# B&R Automation Studio project MM_movim_manuale (part 2)

```c
		if (inst->gs.st_ninfo == 0)																						/* if returned value ok...		*/
		{
			VAL_TO_ASCII(inst->gs.data_typ, inst->gs.ascii_value, inst->gs.var_addr);									/* convert from num to ascii value	*/

			strcpy ( (USINT *)inst->mem_part_all.mem + inst->offset, &inst->gs.name[0]);
			inst->offset = strlen((USINT *) inst->mem_part_all.mem);													/* calculate actual buffer legth	*/
			BUFFER(inst->offset) = inst->chr_separ;																		/* put char separator 			*/
			inst->offset = inst->offset + 1;																			/* calculate actual buffer legth	*/

			inst->get_comm.enable = 1;																					/* enable fub				*/
			Rec_get_comm(&inst->get_comm);																				/* call fub					*/

			if ((inst->get_comm.status == 0) || (inst->get_comm.status == 1))											/* if status ok...			*/
			{
				strcpy ( (USINT *)inst->mem_part_all.mem + inst->offset, &inst->get_comm.comm[0]);						/* ...copy comment			*/
				inst->offset = strlen((USINT *) inst->mem_part_all.mem);												/* calculate actual buffer legth	*/
				BUFFER(inst->offset) = inst->chr_separ;																	/* put char separator 			*/
				inst->offset = inst->offset + 1;																		/* calculate actual buffer legth	*/
			}
			else																										/* if error occurred...			*/
			{
				SET_ERROR(inst->get_comm.status);																		/* ... go to error step			*/
			}
			strcpy ( (USINT *)inst->mem_part_all.mem + inst->offset, inst->gs.ascii_value);								/* copy value (in ascii format)	*/
			inst->offset = strlen((USINT *) inst->mem_part_all.mem);													/* calculate actual buffer legth	*/
			BUFFER(inst->offset    ) = 13;																				/* put carriage return 			*/
			BUFFER(inst->offset + 1) = 10; 																				/* put line feed 				*/
 			inst->offset = inst->offset = inst->offset + 2;																/* calculate actual buffer legth	*/

			memset(&inst->gs.ascii_value, 0, sizeof (inst->gs.ascii_value));											/* reset ascii value buffer		*/

			if (inst->gs.dim[inst->gs.idx_lev] > 1)																		/* if dim > 0 it's an array... 	*/
			{
				clear(&inst->gs.name[0], '[');																			/* ...then delete square brackets 	*/
			}
			if (inst->gs.cnt_dim[inst->gs.idx_lev] < inst->gs.dim[inst->gs.idx_lev] )      								/* if not last element of array... 	*/
			{
				inst->gs.cnt_dim[inst->gs.idx_lev]++;																	/* ...increment index-counter		*/
			}

			for (inst->k = inst->gs.idx_lev;  (inst->gs.cnt_dim[inst->k] == inst->gs.dim[inst->k] && (inst->gs.idx_lev > 0) ); inst->k--)
			{
			 	if (inst->gs.flag_arr_str[inst->k - 1] == 1)															/* if it's an array of structures...*/
				{
					clear(&inst->gs.name[0], '[');																		/* ...delete square brackets		*/
					inst->gs.cnt_arr_str[inst->k-1]++;																	/* increment array of struct counter*/
					if (inst->gs.cnt_arr_str[inst->k-1] >= inst->gs.dim[inst->k - 1] )									/* if array of struct's last element*/
					{
						inst->gs.cnt_arr_str[inst->k-1] = 0;															/* ... reset counter			*/
					}
				}
				else																									/* if field isn't array of structs..*/
				{
					clear(&inst->gs.name[0], '.');																		/* ..delete field name			*/
				}
				inst->gs.cnt_dim[inst->k] = 0;																			/* reset counter for this level	*/
				inst->gs.cnt_dim[inst->k-1] ++;																			/* go ahead for previous level	*/
				inst->gs.idx_lev--;																						/* decrement level 			*/
			}

			if ((inst->gs.idx_lev == 0) &&(inst->gs.cnt_dim[0] == inst->gs.dim[0]))										/* this is the end-condition 		*/
			{
				for (inst->k = 0; inst->k < DEEP_STR; inst->k++)														/* scan all struct (tree)		*/
				{
					inst->gs.cnt_dim[inst->k] = 0;																		/* reset counters about dimensions	*/
					inst->gs.dim[inst->k]     = 0;																		/* reset dimensions			*/
				}
				inst->step = STEP_WST_WRITE_DATA;																		/* ...go again to previous step	*/
			}
			else																										/* if write procedure not finished..*/
			{
				inst->step = STEP_WST_INFO_DATA;																		/* ...go again to previous step	*/
			}
		}
		else																											/* if error occurred...			*/
		{
			SET_ERROR(inst->gs.st_ninfo);																				/* ...go to error step			*/
		}
	}
	else																												/* if error occurred...			*/
	{
	 	SET_ERROR(inst->gs.ret_pvixgetadr);																				/* ...go to error step			*/
	}

} /* end Write_data() */
```

#### Recipe.fun
```iecst
FUNCTION_BLOCK Rec_get_comm
VAR
		step	:USINT;
		k	:UDINT;
		j	:UDINT;
		start	:UDINT;
		do_info	:DatObjInfo;
		count_comm	:UDINT;
		prevstep	:USINT;
	END_VAR
	VAR_INPUT
		enable	:BOOL;
	END_VAR
	VAR_OUTPUT
		comm	:STRING[45];
		status	:UINT;
	END_VAR
END_FUNCTION_BLOCK
FUNCTION_BLOCK Rec_Write
VAR
		overw	:USINT;
		recipecsv	:STRING[24];
		chr_separ	:USINT;
		firstrow_written	:BOOL;
		step	:USINT;
		k	:UDINT;
		fileio_id	:UDINT;
		offset	:UDINT;
		gs	:gs_typ;
		get_comm	:Rec_get_comm;
		FOpen	:FileOpen;
		FCreate	:FileCreate;
		FClose	:FileClose;
		FWrite	:FileWrite;
		FDelete	:FileDelete;
		get_sys_err	:UINT;
		prevstep	:USINT;
		repeat_switch	:USINT;
		mem_part_all	:AsMemPartAlloc;
		mem_allocated	:BOOL;
		mem_part_free	:AsMemPartFree;
		limit_repeat_cntr	:USINT;
		tmp_status	:UINT;
	END_VAR
	VAR_INPUT
		enable	:BOOL;
		structure	:STRING[15];
		recipe	:STRING[20];
		ident	:UDINT;
		speed_option	:BOOL;
	END_VAR
	VAR_OUTPUT
		status	:UINT;
		msg_err	:STRING[80];
	END_VAR
END_FUNCTION_BLOCK
FUNCTION_BLOCK Rec_NameRead
VAR
		step	:USINT;
		set_device	:USINT;
		DInfo	:DirInfo;
		DRead	:DirRead;
		ReadData	:fiDIR_READ_DATA;
		get_sys_err	:UINT;
		prevstep	:USINT;
		len_name	:UINT;
		file_counter	:UDINT;
		tot_files	:UDINT;
		not_valid_csv	:USINT;
	END_VAR
	VAR_INPUT
		enable	:BOOL;
	END_VAR
	VAR_OUTPUT
		status	:UINT;
		msg_err	:STRING[80];
		recipe	:STRING[20];
		nr_csv_read	:UDINT;
	END_VAR
END_FUNCTION_BLOCK
FUNCTION_BLOCK Rec_Import
VAR
		step	:USINT;
		get_sys_err	:UINT;
		prevstep	:UINT;
		recipecsv	:STRING[24];
		FCopy	:FileCopy;
	END_VAR
	VAR_INPUT
		enable	:BOOL;
		recipe	:STRING[20];
	END_VAR
	VAR_OUTPUT
		status	:UINT;
		msg_err	:STRING[80];
	END_VAR
END_FUNCTION_BLOCK
FUNCTION_BLOCK Rec_Imp_All
VAR
		recipe	:STRING[260];
		read_name	:Rec_NameRead;
		rec_imp	:Rec_Import;
		step	:USINT;
		get_sys_err	:UINT;
		prevstep	:USINT;
	END_VAR
	VAR_INPUT
		enable	:BOOL;
	END_VAR
	VAR_OUTPUT
		status	:UINT;
		msg_err	:STRING[80];
		nr_csv_imported	:UDINT;
		recipe_imp	:STRING[80];
	END_VAR
END_FUNCTION_BLOCK
FUNCTION_BLOCK Rec_Export
VAR
		step	:USINT;
		get_sys_err	:UINT;
		prevstep	:UINT;
		recipecsv	:STRING[24];
		FCopy	:FileCopy;
	END_VAR
	VAR_INPUT
		enable	:BOOL;
		recipe	:STRING[20];
	END_VAR
	VAR_OUTPUT
		status	:UINT;
		msg_err	:STRING[80];
	END_VAR
END_FUNCTION_BLOCK
FUNCTION_BLOCK Rec_Exp_All
VAR
		recipe	:STRING[260];
		read_name	:Rec_NameRead;
		rec_exp	:Rec_Export;
		step	:USINT;
		get_sys_err	:UINT;
		prevstep	:USINT;
	END_VAR
	VAR_INPUT
		enable	:BOOL;
	END_VAR
	VAR_OUTPUT
		status	:UINT;
		msg_err	:STRING[80];
	END_VAR
END_FUNCTION_BLOCK
FUNCTION_BLOCK Rec_Upload
VAR
		recipecsv	:STRING[24];
		step	:USINT;
		offset	:UDINT;
		k	:UDINT;
		j	:UDINT;
		ascii_infile	:ARRAY [0..21] OF USINT;
		gs	:gs_typ;
		FOpen	:FileOpen;
		FRead	:FileRead;
		FClose	:FileClose;
		get_sys_err	:UINT;
		repeat_switch	:USINT;
		prevstep	:USINT;
		mem_part_all	:AsMemPartAlloc;
		mem_allocated	:BOOL;
		mem_part_free	:AsMemPartFree;
		limit	:USINT;
		tmp_status	:UINT;
	END_VAR
	VAR_INPUT
		enable	:BOOL;
		structure	:STRING[15];
		recipe	:STRING[20];
		ident	:UDINT;
		speed_option	:BOOL;
	END_VAR
	VAR_OUTPUT
		status	:UINT;
		msg_err	:STRING[80];
	END_VAR
END_FUNCTION_BLOCK
FUNCTION_BLOCK Rec_Delete
VAR
		recipecsv	:STRING[24];
		step	:USINT;
		FDelete	:FileDelete;
		get_sys_err	:UINT;
		prevstep	:USINT;
	END_VAR
	VAR_INPUT
		enable	:BOOL;
		recipe	:STRING[20];
	END_VAR
	VAR_OUTPUT
		status	:UINT;
		msg_err	:STRING[80];
	END_VAR
END_FUNCTION_BLOCK
FUNCTION_BLOCK Rec_Init
VAR
		step	:USINT;
		dir_create	:DirCreate;
		prevstep	:USINT;
		mem_part_create	:AsMemPartCreate;
	END_VAR
	VAR_INPUT
		enable	:BOOL;
	END_VAR
	VAR_OUTPUT
		ident	:UDINT;
		status	:UINT;
		msg_err	:STRING[80];
	END_VAR
END_FUNCTION_BLOCK
```

- Visualisation Logical/Visu (not shown)

### Program Logical/Program (ANSIC)

#### Variables.var
```iecst
VAR
	Apertura_T : BOOL;
	Alta_V_TON : TON;
	Ap_TON : TON;
	Ch_TON : TON;
	Alta_velocita_T : BOOL;
	Chiusura_T : BOOL;
END_VAR
```

#### Cyclic.c
```c
#include <bur/plctypes.h>

#ifdef _DEFAULT_INCLUDES
	#include <AsDefault.h>
#endif

#define CONVERT_INT_TO_ANA_1(x, x1, y1, x2, y2)  ( y1 + ( (y2 - y1) / (REAL) (x2 - x1) ) * (x - x1) )

void _CYCLIC ProgramCyclic(void)
{
	glb_io.Ai.oil_pressure_conv           		= (CONVERT_INT_TO_ANA_1(glb_io.Ai.oil_pressure,           		0,  0, 32767, 250));
	glb_io.Ai.p_apertura_conv           		= (CONVERT_INT_TO_ANA_1(glb_io.Ai.p_apertura,           		0,  0, 32767, 250));
	glb_io.Ai.p_chiusura_conv           		= (CONVERT_INT_TO_ANA_1(glb_io.Ai.p_chiusura,           		0,  0, 32767, 250));

	Report.oil_pressure		= glb_io.Ai.oil_pressure_conv;
	Report.p_apertura		= glb_io.Ai.p_apertura_conv;
	Report.p_apertura		= glb_io.Ai.p_chiusura_conv;

	// ritardo attivazione alta velocità //
	if (hmi.cmd.alta_velocita){
		Alta_V_TON.IN = (hmi.cmd.apertura || hmi.cmd.chiusura);
		Alta_V_TON.PT = 1500;
		TON(&Alta_V_TON);
		Alta_velocita_T = Alta_V_TON.Q;
	} else {
		Alta_velocita_T = 0;
	}
	glb_io.out.alta_velocita = Alta_velocita_T;

	// ritardo attivazione apertura //
	Ap_TON.IN = hmi.cmd.apertura;
	Ap_TON.PT = 500;
	TON(&Ap_TON);
	Apertura_T = Ap_TON.Q;

	// ritardo attivazione chiusura //
	Ch_TON.IN = hmi.cmd.chiusura;
	Ch_TON.PT = 500;
	TON(&Ch_TON);
	Chiusura_T = Ch_TON.Q;

	// COMANDI //
	// SCARICO PRESSIONE //
	if (hmi.cmd.chiusura || hmi.cmd.scarico_ap) glb_io.out.Scarico_ap = 1; else glb_io.out.Scarico_ap = 0;
	if (hmi.cmd.apertura || hmi.cmd.scarico_ch) glb_io.out.Scarico_ch = 1; else glb_io.out.Scarico_ch = 0;

	// ALTA PRESSIONE //
	if (Apertura_T || Chiusura_T || hmi.cmd.lame_fisse_close || hmi.cmd.lame_fisse_open || hmi.cmd.lame_mobili_close
		|| hmi.cmd.lame_mobili_open || hmi.cmd.martinetti_close || hmi.cmd.martinetti_open || hmi.cmd.pedana_dw || hmi.cmd.pedana_up)
	{
		glb_io.out.alta_pressione	= 1;
	} else {
		glb_io.out.alta_pressione	= 0;
	}
	// APERTURA //
	if ((Apertura_T || hmi.cmd.lame_fisse_open || hmi.cmd.lame_mobili_open || hmi.cmd.martinetti_open || hmi.cmd.pedana_up) && (!glb_io.out.chiusura))
	{
		glb_io.out.apertura			= 1;
	} else {
		glb_io.out.apertura			= 0;
	}
	// CHIUSURA //
	if ((Chiusura_T || hmi.cmd.lame_fisse_close || hmi.cmd.lame_mobili_close || hmi.cmd.martinetti_close || hmi.cmd.pedana_dw) && (!glb_io.out.apertura))
	{
		glb_io.out.chiusura			= 1;
	} else {
		glb_io.out.chiusura			= 0;
	}

	// HMI //

	if (hmi.cmd.hmi_oil_control_en){
		oil_control_enable		= 1;
		hmi.cmd.hmi_oil_control_hide	= 0;
	}else {
		oil_control_enable		= 0;
		hmi.cmd.hmi_oil_control_hide 	= 1;
	}

	// CONTROLLO PRESSIONI //
	if (oil_control_enable == 1) {

		// stacco le valvole 41 e 42 se la pressione è troppo alta
		if (glb_io.Ai.oil_pressure_conv >= hmi.inp.MAX_OIL_PRESSURE) {
			glb_io.out.cut_pessure = 1;
		} else if (glb_io.Ai.oil_pressure_conv < hmi.inp.MAX_OIL_PRESSURE - 5) {
			glb_io.out.cut_pessure = 0;
		}
		// stacco pressione se il trasduttore non legge
		if (glb_io.Ai.oil_pressure_conv <= -1) glb_io.out.cut_pessure = 1;

		if (glb_io.out.cut_pessure){
			glb_io.out.alta_pressione	= 0;
			glb_io.out.alta_velocita	= 0;
		}

		if(hmi.cmd.lame_fisse_close){
			if (glb_io.Ai.p_chiusura_conv >= hmi.inp.MAX_OIL_FIX_BLADE_C) {
				glb_io.out.chiusura			= 0;
				glb_io.out.alta_pressione	= 0;
			} else if (glb_io.Ai.p_chiusura_conv < hmi.inp.MAX_OIL_FIX_BLADE_C - 5) {
				//				glb_io.out.chiusura			= 0;
			}

		}else if(hmi.cmd.lame_mobili_close){
			if (glb_io.Ai.p_chiusura_conv >= hmi.inp.MAX_OIL_MOV_BLADE_C) {
				glb_io.out.chiusura			= 0;
				glb_io.out.alta_pressione	= 0;
			} else if (glb_io.Ai.p_chiusura_conv < hmi.inp.MAX_OIL_MOV_BLADE_C - 5) {
				//				glb_io.out.chiusura			= 0;
			}

		}else if(hmi.cmd.martinetti_close){
			if (glb_io.Ai.p_chiusura_conv >= hmi.inp.MAX_OIL_JACK_C) {
				glb_io.out.chiusura			= 0;
				glb_io.out.alta_pressione	= 0;
			} else if (glb_io.Ai.p_chiusura_conv < hmi.inp.MAX_OIL_JACK_C - 5) {
				//				glb_io.out.chiusura			= 0;
			}

		}else if(hmi.cmd.pedana_dw){
			if (glb_io.Ai.p_chiusura_conv >= hmi.inp.MAX_OIL_PEDANA_DW) {
				glb_io.out.chiusura			= 0;
				glb_io.out.alta_pressione	= 0;
			} else if (glb_io.Ai.p_chiusura_conv < hmi.inp.MAX_OIL_PEDANA_DW - 5) {
				//				glb_io.out.chiusura			= 0;
			}

		}else if(hmi.cmd.pedana_up){
			if (glb_io.Ai.p_apertura_conv >= hmi.inp.MAX_OIL_PEDANA_UP) {
				glb_io.out.apertura			= 0;
				glb_io.out.alta_pressione	= 0;
			} else if (glb_io.Ai.p_apertura_conv < hmi.inp.MAX_OIL_PEDANA_UP - 5) {
				//				glb_io.out.chiusura			= 0;
			}
		}
	}

	REPORT;
}
```

#### Init.c
```c
#include <bur/plctypes.h>

#ifdef _DEFAULT_INCLUDES
	#include <AsDefault.h>
#endif

void _INIT ProgramInit(void)
{
	oil_control_enable 			= 1;
	hmi.cmd.hmi_oil_control_en	= 1;
	REPORT						= 1;
}
```

### Program Logical/clock (IEC)

#### Types.typ
```iecst
TYPE
	Typ_Pos : 	STRUCT
		X : LREAL;
		Y : LREAL;
		Z : LREAL;
	END_STRUCT;
	Typ_P : 	STRUCT
		Pos : Typ_Pos;
	END_STRUCT;
END_TYPE
```

#### Variables.var
```iecst
VAR
	DtSetTime_1 : DTSetTime := (0);
	DtGetTime_1 : DTGetTime := (0);
	DT_0 : DATE_AND_TIME := DT#1970-01-01-00:00:00;
	DT_attuale : DATE_AND_TIME := DT#1970-01-01-00:00:00;
END_VAR
```

#### Cyclic.st
```iecst
PROGRAM _CYCLIC
	(* Insert code here *)
	DtSetTime_1.enable;
	DtSetTime_1();
	//status:=DTGetTime_1.status;
	DtSetTime_1.DT1 := DT_attuale;

	DtGetTime_1.enable:=TRUE;
	DtGetTime_1();
	//status:=DTGetTime_1.status;
	DT_0:=DtGetTime_1.DT1;

	//DT_String := DT_TO_STRING();

	IF P THEN
		dir_create.enable := 1;
		//		dir_create.pName := STRING_TO_UDINT( nome);
		dir_create.pName := ADR(nome);
		//		dir_create.pDevice := STRING_TO_UDINT(directory);
		dir_create.pDevice := ADR(directory);
		dir_create();
		P:=0;
	ELSE
		dir_create.enable := 0;
	END_IF

END_PROGRAM
```

#### Init.st
```iecst
PROGRAM _INIT
	(* Insert code here *)
	bOK := FALSE;
	byStep := 1;
	byErrorLevel := 0;
	strDevice       := 'HARDDISK';
	strFile         := 'TestFile';
	(* Initialize read and write data *)
	FOR i := 0 TO 99 DO
		byWriteData[i]  := i + 1;
		byReadData[i]   := 0;
	END_FOR

END_PROGRAM
```

### Program Logical/Alarm (IEC) - Core Alarm handling

#### Cyclic.ld - Cyclic code
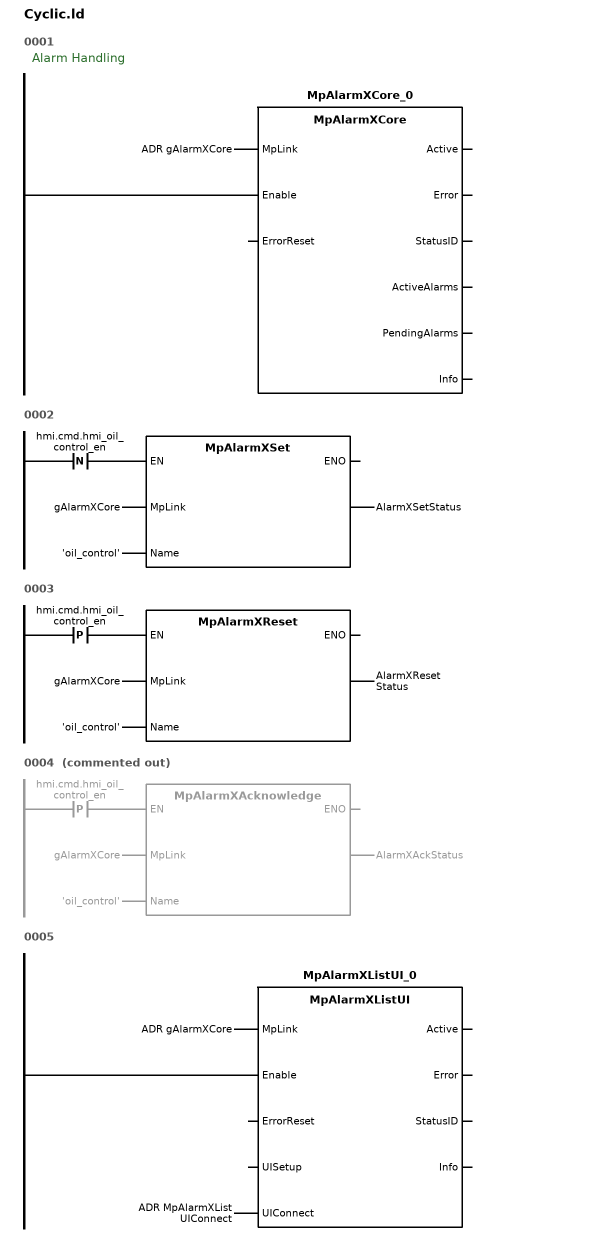
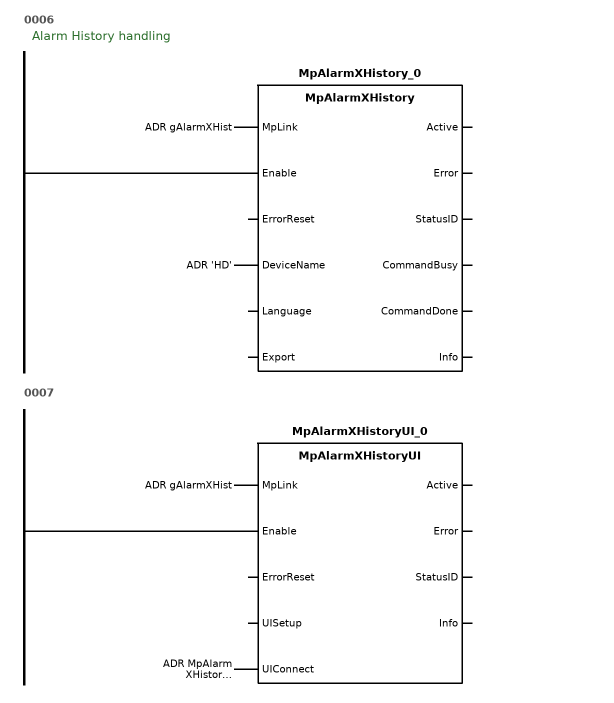
Ladder, written as Structured Text:
```iecst
PROGRAM _CYCLIC
VAR
    _e1 : F_TRIG;
    _e2 : R_TRIG;
    _e3 : R_TRIG;
END_VAR
(* Network 1: Alarm Handling *)
MpAlarmXCore_0(MpLink := ADR(gAlarmXCore), Enable := TRUE);

(* Network 2 *)
_e1(CLK := hmi.cmd.hmi_oil_control_en);
IF _e1.Q THEN AlarmXSetStatus := MpAlarmXSet(MpLink := gAlarmXCore, Name := 'oil_control'); END_IF;

(* Network 3 *)
_e2(CLK := hmi.cmd.hmi_oil_control_en);
IF _e2.Q THEN AlarmXResetStatus := MpAlarmXReset(MpLink := gAlarmXCore, Name := 'oil_control'); END_IF;

(* Network 4 *) (* commented out *)
// _e3(CLK := hmi.cmd.hmi_oil_control_en);
// IF _e3.Q THEN
//     AlarmXAckStatus := MpAlarmXAcknowledge(MpLink := gAlarmXCore, Name := 'oil_control');
// END_IF;

(* Network 5 *)
MpAlarmXListUI_0(MpLink := ADR(gAlarmXCore), Enable := TRUE, UIConnect := ADR(MpAlarmXListUIConnect));

(* Network 6: Alarm History handling *)
MpAlarmXHistory_0(MpLink := ADR(gAlarmXHist), Enable := TRUE, DeviceName := ADR('HD'));

(* Network 7 *)
MpAlarmXHistoryUI_0(MpLink := ADR(gAlarmXHist), Enable := TRUE, UIConnect := ADR(MpAlarmXHistoryUIConnect));
END_PROGRAM
```

#### Variables.var - Local variables
```iecst
VAR
	MpAlarmXHistory_0 : MpAlarmXHistory; (*MpAlarmXHistory instance*)
	MpAlarmXHistoryUI_0 : MpAlarmXHistoryUI := (UISetup:=(AlarmListSize:=9)); (*MpAlarmXHistoryUI instance*)
	MpAlarmXListUI_0 : MpAlarmXListUI := (UISetup:=(AlarmListSize:=9)); (*MpAlarmXList instance*)
	MpAlarmXHistoryUIConnect : MpAlarmXHistoryUIConnectType; (*MpAlarmXHistoryUI UI connection points*)
	MpAlarmXListUIConnect : MpAlarmXListUIConnectType; (*MpAlarmXListUI UI connection points*)
	MpAlarmXCore_0 : MpAlarmXCore; (*MpAlarmXCore instance*)
	AlarmXSetStatus : UDINT;
	AlarmXResetStatus : DINT;
	AlarmXAckStatus : DINT;
	alm_export : BOOL;
END_VAR
```

### Program Logical/Data (IEC) - Core Data recording

#### Cyclic.ld - Cyclic code
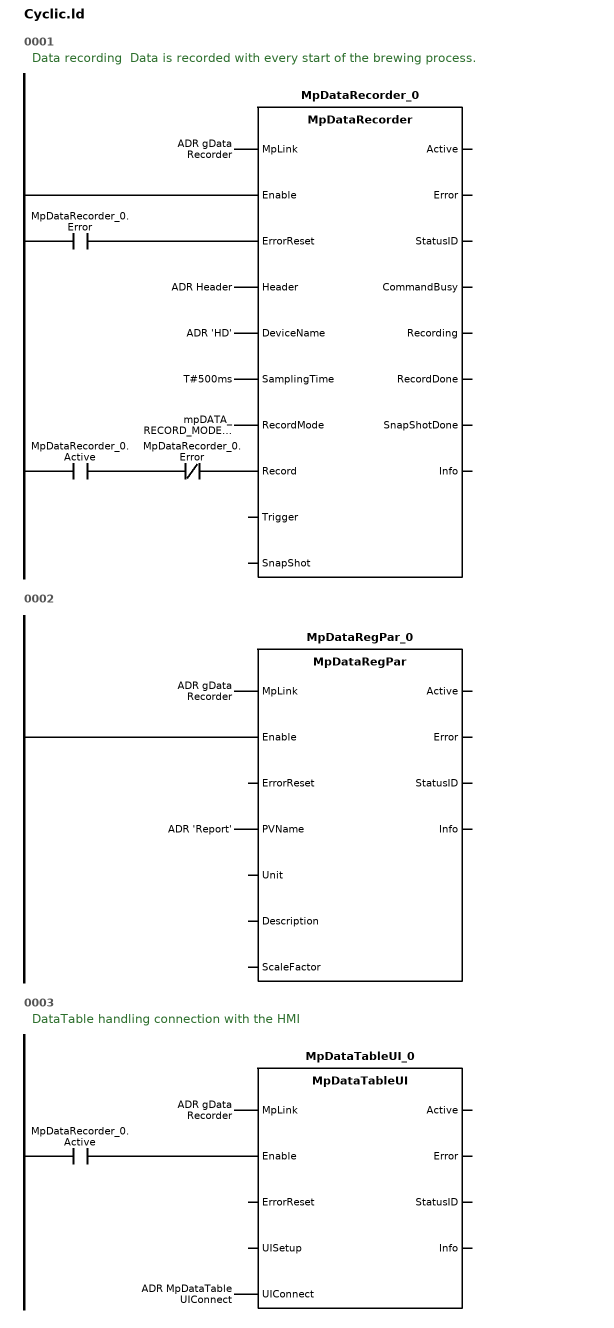
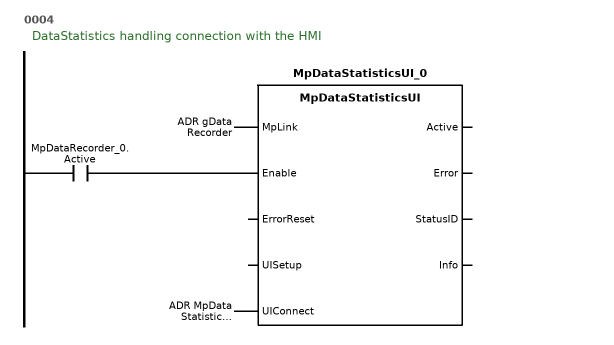
Ladder, written as Structured Text:
```iecst
PROGRAM _CYCLIC
(* Network 1: Data recording  Data is recorded with every start of the brewing process. *)
MpDataRecorder_0(MpLink := ADR(gDataRecorder), Enable := TRUE, ErrorReset := MpDataRecorder_0.Error, Header := ADR(Header), DeviceName := ADR('HD'), SamplingTime := T#500ms, RecordMode := mpDATA_RECORD_MODE_TIME, Record := MpDataRecorder_0.Active AND NOT MpDataRecorder_0.Error);

(* Network 2 *)
MpDataRegPar_0(MpLink := ADR(gDataRecorder), Enable := TRUE, PVName := ADR('Report'));

(* Network 3: DataTable handling connection with the HMI *)
MpDataTableUI_0(MpLink := ADR(gDataRecorder), Enable := MpDataRecorder_0.Active, UIConnect := ADR(MpDataTableUIConnect));

(* Network 4: DataStatistics handling connection with the HMI *)
MpDataStatisticsUI_0(MpLink := ADR(gDataRecorder), Enable := MpDataRecorder_0.Active, UIConnect := ADR(MpDataStatisticsUIConnect));
END_PROGRAM
```

#### Init.ld - Init code
Ladder, written as Structured Text:
```iecst
PROGRAM _INIT
(* Network 1 *)
END_PROGRAM
```

#### Variables.var - Local variables
```iecst
VAR
	MpDataRegPar_0 : MpDataRegPar;
	Enable : BOOL := TRUE; (*Enable the component, can be used in the watch window to change the setup*)
	MpDataRecorder_0 : MpDataRecorder := (SamplingTime:=T#500ms); (*MpDataRecorder FUB*)
	Status : DINT := 0; (*Status variable the MpAlarmBasicSet / ResetAlarm functions*)
	MpDataTableUI_0 : MpDataTableUI := (UISetup:=(ValueListSize:=10,PVListSize:=5)); (*MpDataTableUI FUB*)
	MpDataTableUIConnect : MpDataTableUIConnectType; (*MpDataTableUI connection datapoints*)
	Header : MpDataRecorderHeaderType := (Name:='Report Pressioni',Description:='Campionamento delle pressioni ogni 0,5s'); (*Header description for UI components*)
	MpDataStatisticsUI_0 : MpDataStatisticsUI := (UISetup:=(PVListSize:=6)); (*MpDataStatisticsUI FUB*)
	MpDataStatisticsUIConnect : MpDataStatisticsUIConnectType; (*MpDataStatisticsUI connection datapoints*)
END_VAR
```

- Visualisation Logical/Visu_Resized (not shown)
